REGION Network 132: BA015 Interface Data
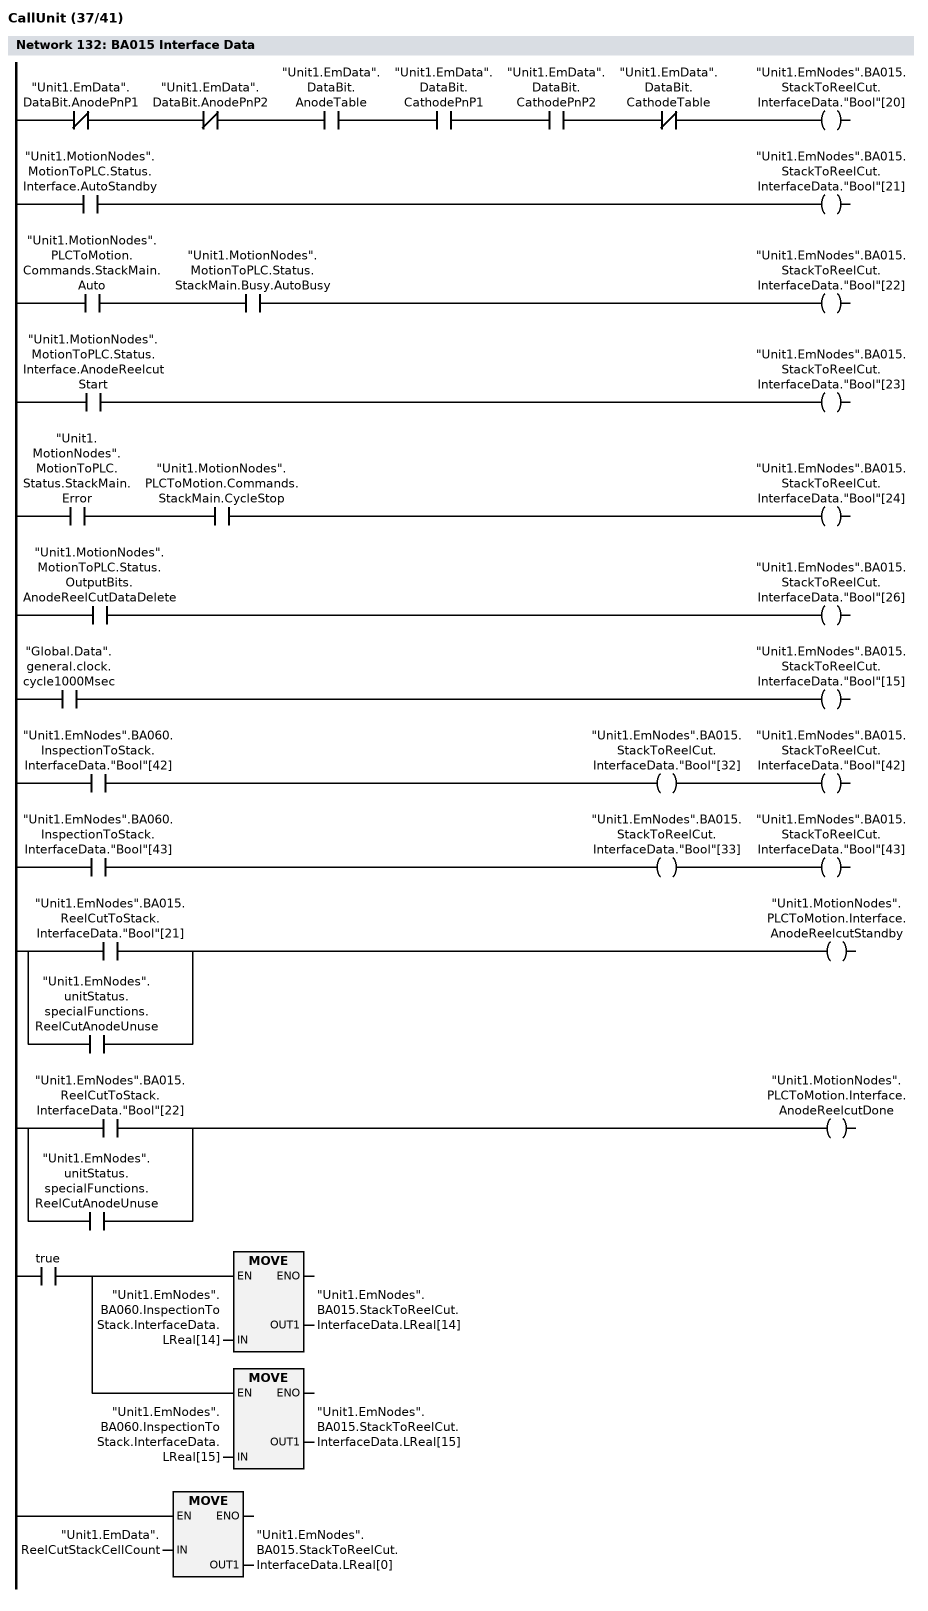
   RUNG wire#powerrail
      I_Contact( "Unit1.EmData".DataBit.AnodePnP1 )
      I_Contact( "Unit1.EmData".DataBit.AnodePnP2 )
      Contact( "Unit1.EmData".DataBit.AnodeTable )
      Contact( "Unit1.EmData".DataBit.CathodePnP1 )
      Contact( "Unit1.EmData".DataBit.CathodePnP2 )
      I_Contact( "Unit1.EmData".DataBit.CathodeTable )
      Coil( "Unit1.EmNodes".BA015.StackToReelCut.InterfaceData."Bool"[20] )
   END_RUNG
   RUNG wire#powerrail
      Contact( "Unit1.MotionNodes".MotionToPLC.Status.Interface.AutoStandby )
      Coil( "Unit1.EmNodes".BA015.StackToReelCut.InterfaceData."Bool"[21] )
   END_RUNG
   RUNG wire#powerrail
      Contact( "Unit1.MotionNodes".PLCToMotion.Commands.StackMain.Auto )
      Contact( "Unit1.MotionNodes".MotionToPLC.Status.StackMain.Busy.AutoBusy )
      Coil( "Unit1.EmNodes".BA015.StackToReelCut.InterfaceData."Bool"[22] )
   END_RUNG
   RUNG wire#powerrail
      Contact( "Unit1.MotionNodes".MotionToPLC.Status.Interface.AnodeReelcutStart )
      Coil( "Unit1.EmNodes".BA015.StackToReelCut.InterfaceData."Bool"[23] )
   END_RUNG
   RUNG wire#powerrail
      Contact( "Unit1.MotionNodes".MotionToPLC.Status.StackMain.Error )
      Contact( "Unit1.MotionNodes".PLCToMotion.Commands.StackMain.CycleStop )
      Coil( "Unit1.EmNodes".BA015.StackToReelCut.InterfaceData."Bool"[24] )
   END_RUNG
   RUNG wire#powerrail
      Contact( "Unit1.MotionNodes".MotionToPLC.Status.OutputBits.AnodeReelCutDataDelete )
      Coil( "Unit1.EmNodes".BA015.StackToReelCut.InterfaceData."Bool"[26] )
   END_RUNG
   RUNG wire#powerrail
      Contact( "Global.Data".general.clock.cycle1000Msec )
      Coil( "Unit1.EmNodes".BA015.StackToReelCut.InterfaceData."Bool"[15] )
   END_RUNG
   RUNG wire#powerrail
      Contact( "Unit1.EmNodes".BA060.InspectionToStack.InterfaceData."Bool"[42] )
      Coil( "Unit1.EmNodes".BA015.StackToReelCut.InterfaceData."Bool"[32] )
      Coil( "Unit1.EmNodes".BA015.StackToReelCut.InterfaceData."Bool"[42] )
   END_RUNG
   RUNG wire#powerrail
      Contact( "Unit1.EmNodes".BA060.InspectionToStack.InterfaceData."Bool"[43] )
      Coil( "Unit1.EmNodes".BA015.StackToReelCut.InterfaceData."Bool"[33] )
      Coil( "Unit1.EmNodes".BA015.StackToReelCut.InterfaceData."Bool"[43] )
   END_RUNG
   RUNG wire#powerrail
      Contact( "Unit1.EmNodes".BA015.ReelCutToStack.InterfaceData."Bool"[21] )
      wire#w1
      Coil( "Unit1.MotionNodes".PLCToMotion.Interface.AnodeReelcutStandby )
   END_RUNG
   RUNG wire#powerrail
      Contact( "Unit1.EmNodes".unitStatus.specialFunctions.ReelCutAnodeUnuse )
   END_RUNG wire#w1
   RUNG wire#powerrail
      Contact( "Unit1.EmNodes".BA015.ReelCutToStack.InterfaceData."Bool"[22] )
      wire#w2
      Coil( "Unit1.MotionNodes".PLCToMotion.Interface.AnodeReelcutDone )
   END_RUNG
   RUNG wire#powerrail
      Contact( "Unit1.EmNodes".unitStatus.specialFunctions.ReelCutAnodeUnuse )
   END_RUNG wire#w2
   RUNG wire#powerrail
      Contact( true )
      wire#w3
      Move(in := "Unit1.EmNodes".BA060.InspectionToStack.InterfaceData.LReal[14], out1 => "Unit1.EmNodes".BA015.StackToReelCut.InterfaceData.LReal[14])
   END_RUNG
   RUNG wire#w3
      Move(in := "Unit1.EmNodes".BA060.InspectionToStack.InterfaceData.LReal[15], out1 => "Unit1.EmNodes".BA015.StackToReelCut.InterfaceData.LReal[15])
   END_RUNG
   RUNG wire#powerrail
      Move(in := "Unit1.EmData".ReelCutStackCellCount, out1 => "Unit1.EmNodes".BA015.StackToReelCut.InterfaceData.LReal[0])
   END_RUNG
   // the same network as SCL:
   "Unit1.EmNodes".BA015.StackToReelCut.InterfaceData."Bool"[20] := NOT "Unit1.EmData".DataBit.AnodePnP1 AND NOT "Unit1.EmData".DataBit.AnodePnP2 AND "Unit1.EmData".DataBit.AnodeTable AND "Unit1.EmData".DataBit.CathodePnP1 AND "Unit1.EmData".DataBit.CathodePnP2 AND NOT "Unit1.EmData".DataBit.CathodeTable;
   "Unit1.EmNodes".BA015.StackToReelCut.InterfaceData."Bool"[21] := "Unit1.MotionNodes".MotionToPLC.Status.Interface.AutoStandby;
   "Unit1.EmNodes".BA015.StackToReelCut.InterfaceData."Bool"[22] := "Unit1.MotionNodes".PLCToMotion.Commands.StackMain.Auto AND "Unit1.MotionNodes".MotionToPLC.Status.StackMain.Busy.AutoBusy;
   "Unit1.EmNodes".BA015.StackToReelCut.InterfaceData."Bool"[23] := "Unit1.MotionNodes".MotionToPLC.Status.Interface.AnodeReelcutStart;
   "Unit1.EmNodes".BA015.StackToReelCut.InterfaceData."Bool"[24] := "Unit1.MotionNodes".MotionToPLC.Status.StackMain.Error AND "Unit1.MotionNodes".PLCToMotion.Commands.StackMain.CycleStop;
   "Unit1.EmNodes".BA015.StackToReelCut.InterfaceData."Bool"[26] := "Unit1.MotionNodes".MotionToPLC.Status.OutputBits.AnodeReelCutDataDelete;
   "Unit1.EmNodes".BA015.StackToReelCut.InterfaceData."Bool"[15] := "Global.Data".general.clock.cycle1000Msec;
   "Unit1.EmNodes".BA015.StackToReelCut.InterfaceData."Bool"[32] := "Unit1.EmNodes".BA060.InspectionToStack.InterfaceData."Bool"[42];
   "Unit1.EmNodes".BA015.StackToReelCut.InterfaceData."Bool"[42] := "Unit1.EmNodes".BA060.InspectionToStack.InterfaceData."Bool"[42];
   "Unit1.EmNodes".BA015.StackToReelCut.InterfaceData."Bool"[33] := "Unit1.EmNodes".BA060.InspectionToStack.InterfaceData."Bool"[43];
   "Unit1.EmNodes".BA015.StackToReelCut.InterfaceData."Bool"[43] := "Unit1.EmNodes".BA060.InspectionToStack.InterfaceData."Bool"[43];
   "Unit1.MotionNodes".PLCToMotion.Interface.AnodeReelcutStandby := "Unit1.EmNodes".BA015.ReelCutToStack.InterfaceData."Bool"[21] OR "Unit1.EmNodes".unitStatus.specialFunctions.ReelCutAnodeUnuse;
   "Unit1.MotionNodes".PLCToMotion.Interface.AnodeReelcutDone := "Unit1.EmNodes".BA015.ReelCutToStack.InterfaceData."Bool"[22] OR "Unit1.EmNodes".unitStatus.specialFunctions.ReelCutAnodeUnuse;
   IF true THEN
       "Unit1.EmNodes".BA015.StackToReelCut.InterfaceData.LReal[14] := "Unit1.EmNodes".BA060.InspectionToStack.InterfaceData.LReal[14];
       "Unit1.EmNodes".BA015.StackToReelCut.InterfaceData.LReal[15] := "Unit1.EmNodes".BA060.InspectionToStack.InterfaceData.LReal[15];
   END_IF;
   "Unit1.EmNodes".BA015.StackToReelCut.InterfaceData.LReal[0] := "Unit1.EmData".ReelCutStackCellCount;
END_REGION

REGION Network 133: Stack To ReelCut BA015 Unit Status
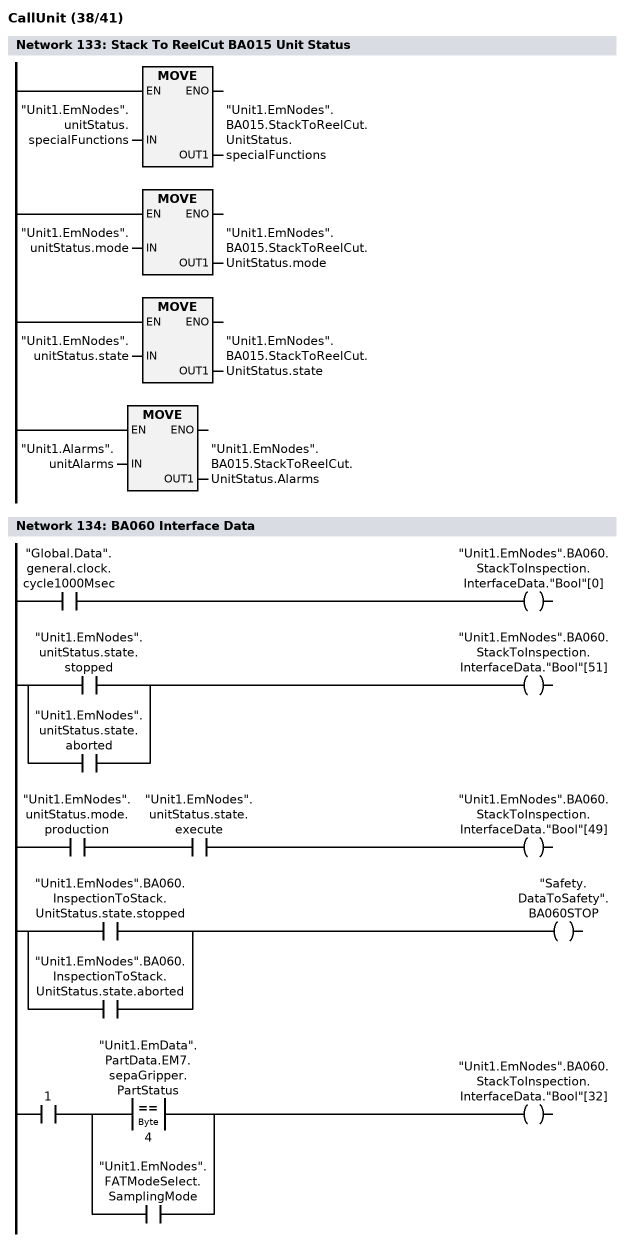
   RUNG wire#powerrail
      Move(in := "Unit1.EmNodes".unitStatus.specialFunctions, out1 => "Unit1.EmNodes".BA015.StackToReelCut.UnitStatus.specialFunctions)
   END_RUNG
   RUNG wire#powerrail
      Move(in := "Unit1.EmNodes".unitStatus.mode, out1 => "Unit1.EmNodes".BA015.StackToReelCut.UnitStatus.mode)
   END_RUNG
   RUNG wire#powerrail
      Move(in := "Unit1.EmNodes".unitStatus.state, out1 => "Unit1.EmNodes".BA015.StackToReelCut.UnitStatus.state)
   END_RUNG
   RUNG wire#powerrail
      Move(in := "Unit1.Alarms".unitAlarms, out1 => "Unit1.EmNodes".BA015.StackToReelCut.UnitStatus.Alarms)
   END_RUNG
   // the same network as SCL:
   "Unit1.EmNodes".BA015.StackToReelCut.UnitStatus.specialFunctions := "Unit1.EmNodes".unitStatus.specialFunctions;
   "Unit1.EmNodes".BA015.StackToReelCut.UnitStatus.mode := "Unit1.EmNodes".unitStatus.mode;
   "Unit1.EmNodes".BA015.StackToReelCut.UnitStatus.state := "Unit1.EmNodes".unitStatus.state;
   "Unit1.EmNodes".BA015.StackToReelCut.UnitStatus.Alarms := "Unit1.Alarms".unitAlarms;
END_REGION

REGION Network 134: BA060 Interface Data
   RUNG wire#powerrail
      Contact( "Global.Data".general.clock.cycle1000Msec )
      Coil( "Unit1.EmNodes".BA060.StackToInspection.InterfaceData."Bool"[0] )
   END_RUNG
   RUNG wire#powerrail
      Contact( "Unit1.EmNodes".unitStatus.state.stopped )
      wire#w1
      Coil( "Unit1.EmNodes".BA060.StackToInspection.InterfaceData."Bool"[51] )
   END_RUNG
   RUNG wire#powerrail
      Contact( "Unit1.EmNodes".unitStatus.state.aborted )
   END_RUNG wire#w1
   RUNG wire#powerrail
      Contact( "Unit1.EmNodes".unitStatus.mode.production )
      Contact( "Unit1.EmNodes".unitStatus.state.execute )
      Coil( "Unit1.EmNodes".BA060.StackToInspection.InterfaceData."Bool"[49] )
   END_RUNG
   RUNG wire#powerrail
      Contact( "Unit1.EmNodes".BA060.InspectionToStack.UnitStatus.state.stopped )
      wire#w2
      Coil( "Safety.DataToSafety".BA060STOP )
   END_RUNG
   RUNG wire#powerrail
      Contact( "Unit1.EmNodes".BA060.InspectionToStack.UnitStatus.state.aborted )
   END_RUNG wire#w2
   RUNG wire#powerrail
      Contact( 1 )
      wire#w3
      { S7_Templates := "SrcType := Byte" } EQ_Contact(in1 := "Unit1.EmData".PartData.EM7.sepaGripper.PartStatus, in2 := 4)
      wire#w4
      Coil( "Unit1.EmNodes".BA060.StackToInspection.InterfaceData."Bool"[32] )
   END_RUNG
   RUNG wire#w3
      Contact( "Unit1.EmNodes".FATModeSelect.SamplingMode )
   END_RUNG wire#w4
   // the same network as SCL:
   "Unit1.EmNodes".BA060.StackToInspection.InterfaceData."Bool"[0] := "Global.Data".general.clock.cycle1000Msec;
   "Unit1.EmNodes".BA060.StackToInspection.InterfaceData."Bool"[51] := "Unit1.EmNodes".unitStatus.state.stopped OR "Unit1.EmNodes".unitStatus.state.aborted;
   "Unit1.EmNodes".BA060.StackToInspection.InterfaceData."Bool"[49] := "Unit1.EmNodes".unitStatus.mode.production AND "Unit1.EmNodes".unitStatus.state.execute;
   "Safety.DataToSafety".BA060STOP := "Unit1.EmNodes".BA060.InspectionToStack.UnitStatus.state.stopped OR "Unit1.EmNodes".BA060.InspectionToStack.UnitStatus.state.aborted;
   "Unit1.EmNodes".BA060.StackToInspection.InterfaceData."Bool"[32] := 1 AND (("Unit1.EmData".PartData.EM7.sepaGripper.PartStatus = 4) OR "Unit1.EmNodes".FATModeSelect.SamplingMode);
END_REGION

REGION Network 135: Stack To Insp BA060 specialFuctions
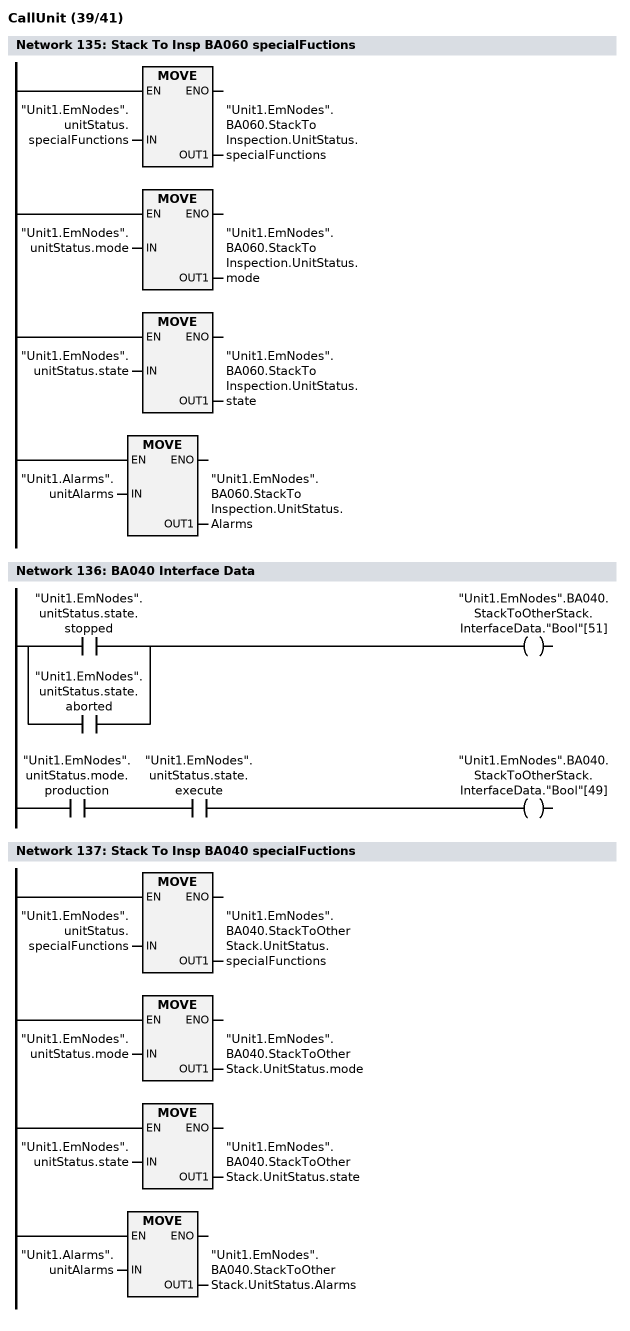
   RUNG wire#powerrail
      Move(in := "Unit1.EmNodes".unitStatus.specialFunctions, out1 => "Unit1.EmNodes".BA060.StackToInspection.UnitStatus.specialFunctions)
   END_RUNG
   RUNG wire#powerrail
      Move(in := "Unit1.EmNodes".unitStatus.mode, out1 => "Unit1.EmNodes".BA060.StackToInspection.UnitStatus.mode)
   END_RUNG
   RUNG wire#powerrail
      Move(in := "Unit1.EmNodes".unitStatus.state, out1 => "Unit1.EmNodes".BA060.StackToInspection.UnitStatus.state)
   END_RUNG
   RUNG wire#powerrail
      Move(in := "Unit1.Alarms".unitAlarms, out1 => "Unit1.EmNodes".BA060.StackToInspection.UnitStatus.Alarms)
   END_RUNG
   // the same network as SCL:
   "Unit1.EmNodes".BA060.StackToInspection.UnitStatus.specialFunctions := "Unit1.EmNodes".unitStatus.specialFunctions;
   "Unit1.EmNodes".BA060.StackToInspection.UnitStatus.mode := "Unit1.EmNodes".unitStatus.mode;
   "Unit1.EmNodes".BA060.StackToInspection.UnitStatus.state := "Unit1.EmNodes".unitStatus.state;
   "Unit1.EmNodes".BA060.StackToInspection.UnitStatus.Alarms := "Unit1.Alarms".unitAlarms;
END_REGION

REGION Network 136: BA040 Interface Data
   RUNG wire#powerrail
      Contact( "Unit1.EmNodes".unitStatus.state.stopped )
      wire#w1
      Coil( "Unit1.EmNodes".BA040.StackToOtherStack.InterfaceData."Bool"[51] )
   END_RUNG
   RUNG wire#powerrail
      Contact( "Unit1.EmNodes".unitStatus.state.aborted )
   END_RUNG wire#w1
   RUNG wire#powerrail
      Contact( "Unit1.EmNodes".unitStatus.mode.production )
      Contact( "Unit1.EmNodes".unitStatus.state.execute )
      Coil( "Unit1.EmNodes".BA040.StackToOtherStack.InterfaceData."Bool"[49] )
   END_RUNG
   // the same network as SCL:
   "Unit1.EmNodes".BA040.StackToOtherStack.InterfaceData."Bool"[51] := "Unit1.EmNodes".unitStatus.state.stopped OR "Unit1.EmNodes".unitStatus.state.aborted;
   "Unit1.EmNodes".BA040.StackToOtherStack.InterfaceData."Bool"[49] := "Unit1.EmNodes".unitStatus.mode.production AND "Unit1.EmNodes".unitStatus.state.execute;
END_REGION

REGION Network 137: Stack To Insp BA040 specialFuctions
   RUNG wire#powerrail
      Move(in := "Unit1.EmNodes".unitStatus.specialFunctions, out1 => "Unit1.EmNodes".BA040.StackToOtherStack.UnitStatus.specialFunctions)
   END_RUNG
   RUNG wire#powerrail
      Move(in := "Unit1.EmNodes".unitStatus.mode, out1 => "Unit1.EmNodes".BA040.StackToOtherStack.UnitStatus.mode)
   END_RUNG
   RUNG wire#powerrail
      Move(in := "Unit1.EmNodes".unitStatus.state, out1 => "Unit1.EmNodes".BA040.StackToOtherStack.UnitStatus.state)
   END_RUNG
   RUNG wire#powerrail
      Move(in := "Unit1.Alarms".unitAlarms, out1 => "Unit1.EmNodes".BA040.StackToOtherStack.UnitStatus.Alarms)
   END_RUNG
   // the same network as SCL:
   "Unit1.EmNodes".BA040.StackToOtherStack.UnitStatus.specialFunctions := "Unit1.EmNodes".unitStatus.specialFunctions;
   "Unit1.EmNodes".BA040.StackToOtherStack.UnitStatus.mode := "Unit1.EmNodes".unitStatus.mode;
   "Unit1.EmNodes".BA040.StackToOtherStack.UnitStatus.state := "Unit1.EmNodes".unitStatus.state;
   "Unit1.EmNodes".BA040.StackToOtherStack.UnitStatus.Alarms := "Unit1.Alarms".unitAlarms;
END_REGION

REGION Network 138: Q-DAS
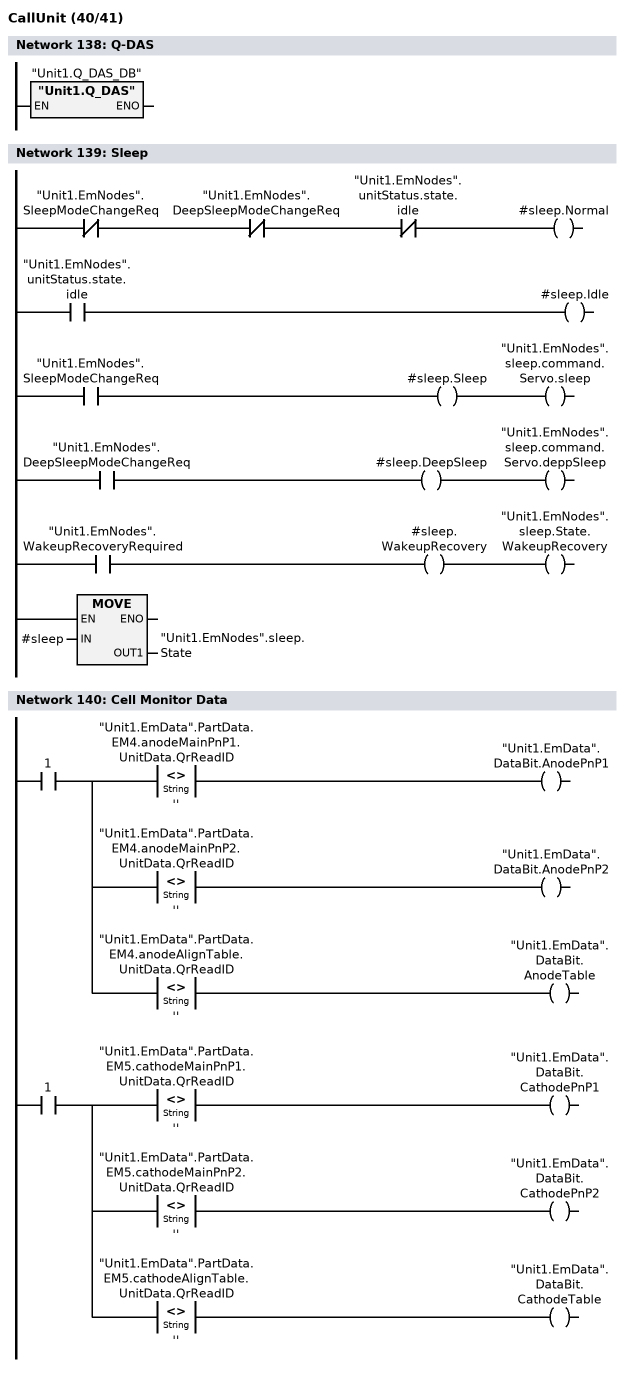
   RUNG wire#powerrail
      "Unit1.Q_DAS_DB"()
   END_RUNG
   // the same network as SCL:
   "Unit1.Q_DAS_DB"();   // "Unit1.Q_DAS"
END_REGION

REGION Network 139: Sleep
   RUNG wire#powerrail
      I_Contact( "Unit1.EmNodes".SleepModeChangeReq )
      I_Contact( "Unit1.EmNodes".DeepSleepModeChangeReq )
      I_Contact( "Unit1.EmNodes".unitStatus.state.idle )
      Coil( #sleep.Normal )
   END_RUNG
   RUNG wire#powerrail
      Contact( "Unit1.EmNodes".unitStatus.state.idle )
      Coil( #sleep.Idle )
   END_RUNG
   RUNG wire#powerrail
      Contact( "Unit1.EmNodes".SleepModeChangeReq )
      Coil( #sleep.Sleep )
      Coil( "Unit1.EmNodes".sleep.command.Servo.sleep )
   END_RUNG
   RUNG wire#powerrail
      Contact( "Unit1.EmNodes".DeepSleepModeChangeReq )
      Coil( #sleep.DeepSleep )
      Coil( "Unit1.EmNodes".sleep.command.Servo.deppSleep )
   END_RUNG
   RUNG wire#powerrail
      Contact( "Unit1.EmNodes".WakeupRecoveryRequired )
      Coil( #sleep.WakeupRecovery )
      Coil( "Unit1.EmNodes".sleep.State.WakeupRecovery )
   END_RUNG
   RUNG wire#powerrail
      Move(in := #sleep, out1 => "Unit1.EmNodes".sleep.State)
   END_RUNG
   // the same network as SCL:
   #sleep.Normal := NOT "Unit1.EmNodes".SleepModeChangeReq AND NOT "Unit1.EmNodes".DeepSleepModeChangeReq AND NOT "Unit1.EmNodes".unitStatus.state.idle;
   #sleep.Idle := "Unit1.EmNodes".unitStatus.state.idle;
   #sleep.Sleep := "Unit1.EmNodes".SleepModeChangeReq;
   "Unit1.EmNodes".sleep.command.Servo.sleep := "Unit1.EmNodes".SleepModeChangeReq;
   #sleep.DeepSleep := "Unit1.EmNodes".DeepSleepModeChangeReq;
   "Unit1.EmNodes".sleep.command.Servo.deppSleep := "Unit1.EmNodes".DeepSleepModeChangeReq;
   #sleep.WakeupRecovery := "Unit1.EmNodes".WakeupRecoveryRequired;
   "Unit1.EmNodes".sleep.State.WakeupRecovery := "Unit1.EmNodes".WakeupRecoveryRequired;
   "Unit1.EmNodes".sleep.State := #sleep;
END_REGION

REGION Network 140: Cell Monitor Data
   RUNG wire#powerrail
      Contact( 1 )
      wire#w1
      { S7_Templates := "SrcType := String" } NE_Contact(in1 := "Unit1.EmData".PartData.EM4.anodeMainPnP1.UnitData.QrReadID, in2 := '')
      Coil( "Unit1.EmData".DataBit.AnodePnP1 )
   END_RUNG
   RUNG wire#w1
      { S7_Templates := "SrcType := String" } NE_Contact(in1 := "Unit1.EmData".PartData.EM4.anodeMainPnP2.UnitData.QrReadID, in2 := '')
      Coil( "Unit1.EmData".DataBit.AnodePnP2 )
   END_RUNG
   RUNG wire#w1
      { S7_Templates := "SrcType := String" } NE_Contact(in1 := "Unit1.EmData".PartData.EM4.anodeAlignTable.UnitData.QrReadID, in2 := '')
      Coil( "Unit1.EmData".DataBit.AnodeTable )
   END_RUNG
   RUNG wire#powerrail
      Contact( 1 )
      wire#w2
      { S7_Templates := "SrcType := String" } NE_Contact(in1 := "Unit1.EmData".PartData.EM5.cathodeMainPnP1.UnitData.QrReadID, in2 := '')
      Coil( "Unit1.EmData".DataBit.CathodePnP1 )
   END_RUNG
   RUNG wire#w2
      { S7_Templates := "SrcType := String" } NE_Contact(in1 := "Unit1.EmData".PartData.EM5.cathodeMainPnP2.UnitData.QrReadID, in2 := '')
      Coil( "Unit1.EmData".DataBit.CathodePnP2 )
   END_RUNG
   RUNG wire#w2
      { S7_Templates := "SrcType := String" } NE_Contact(in1 := "Unit1.EmData".PartData.EM5.cathodeAlignTable.UnitData.QrReadID, in2 := '')
      Coil( "Unit1.EmData".DataBit.CathodeTable )
   END_RUNG
   // the same network as SCL:
   "Unit1.EmData".DataBit.AnodePnP1 := 1 AND ("Unit1.EmData".PartData.EM4.anodeMainPnP1.UnitData.QrReadID <> '');
   "Unit1.EmData".DataBit.AnodePnP2 := 1 AND ("Unit1.EmData".PartData.EM4.anodeMainPnP2.UnitData.QrReadID <> '');
   "Unit1.EmData".DataBit.AnodeTable := 1 AND ("Unit1.EmData".PartData.EM4.anodeAlignTable.UnitData.QrReadID <> '');
   "Unit1.EmData".DataBit.CathodePnP1 := 1 AND ("Unit1.EmData".PartData.EM5.cathodeMainPnP1.UnitData.QrReadID <> '');
   "Unit1.EmData".DataBit.CathodePnP2 := 1 AND ("Unit1.EmData".PartData.EM5.cathodeMainPnP2.UnitData.QrReadID <> '');
   "Unit1.EmData".DataBit.CathodeTable := 1 AND ("Unit1.EmData".PartData.EM5.cathodeAlignTable.UnitData.QrReadID <> '');
END_REGION

REGION Network 141: Motion Data
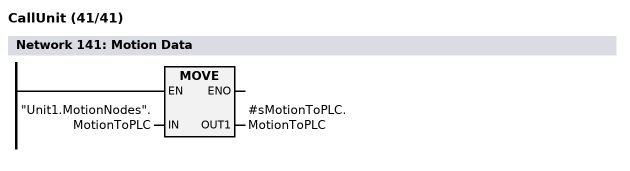
   RUNG wire#powerrail
      Move(in := "Unit1.MotionNodes".MotionToPLC, out1 => #sMotionToPLC.MotionToPLC)
   END_RUNG
   // the same network as SCL:
   #sMotionToPLC.MotionToPLC := "Unit1.MotionNodes".MotionToPLC;
END_REGION
END_FUNCTION_BLOCK
